(* CoDeSys 2.3.9.59 project: ProgettoSFC.pro *)
(* Libraries: STANDARD.LIB, Iecsfc.lib 12.5.98 11:03:00 *)

(* Task configuration *)
TASK Standard (PRIORITY := 0, INTERVAL := T#10ms);
	MAIN
END_TASK

(* Data type *)
TYPE ALTEZZA: (nd_A, basso, alto);
END_TYPE

(* Data type *)
TYPE COLORE: (nd_C, rosso, altro);
END_TYPE

(* Data type *)
TYPE LOCK_INGRESSO_GIOSTRA :
STRUCT
  FlagNastro: BOOL:=FALSE;
  FlagGIostra: BOOL:=FALSE;
  Turno: TURNO;
END_STRUCT
END_TYPE

(* Data type *)
TYPE PEZZO :
STRUCT
	Colore :COLORE;
	Altezza :ALTEZZA;
END_STRUCT
END_TYPE

(* Data type *)
TYPE POSTO :
STRUCT
	Presenza :BOOL;
	Pezzo :PEZZO;
	Ready :BOOL; (*uguale a 1 quando nel posto è terminato il lavoro*)
	Fine_Lavorazione :BOOL;
END_STRUCT
END_TYPE

(* Data type *)
TYPE TURNO : (Giostr, nastro);
END_TYPE

(* POU MAIN, SFC *)
PROGRAM MAIN
VAR

(*Variabili Pistone*)
  Presenza_Pezzo AT %IX0.0: BOOL;
  Pistone_Indietro AT %IX0.4: BOOL;
  Pistone_Avanti AT %IX0.2: BOOL;
  Pistone_On AT %QX0.2: BOOL;

(*Variabili nastro*)
  Nastro_On AT %QX0.0: BOOL;
  Fine_Corsa AT %IX0.6: BOOL;
  NumPeN: INT:= 0;

(*Variabili gestione timers per non creare conflitti tra nastro pistone e giostra*)
  TimerNP: TON;
  Timer_GN: TON;
  Timer_Nastro: TON;
  ResetTimer: BOOL := FALSE;
  AttesaNP: TIME:= t#0.6s;
  Q: BOOL;
  Delay_Pistone: TON;
  Ritardo_Pistone: BOOL;


(*Interfaccia Nastro-Giostra*)
  InserimentoNG: BOOL:=FALSE; (*Il nastro deve mettere a TRUE quando sta inserendo un pezzo all'interno della giostra e a FALSE quando non lo sta facendo*)
  FineInserimentoGN: BOOL;
  NReady: BOOL := TRUE;    (*Vero quando il nastro autorizza il pistone a spingere un nuovo pezzo*)
  GStart: BOOL := TRUE;    (*Vero quando la giostra è autorizzata a girare*)


(*variabili giostra*)
  Movimento_Giostra AT %QX3.4: BOOL;
  Giostra_BUSY AT %IX6.1: BOOL;
  Giostra: ARRAY[0..7] OF POSTO; (*Array che descrive lo stato di tutti i posti della giostra*)
  TEMP: ARRAY[0..7] OF BOOL; (*Array di supporto per verificare delle condizioni su array di 8 elementi*)
  presenza_fine_lav: BOOL; (*Variabile che deve essere settata a TRUE quando tutti i pezzi presenti nella giostra hanno finito la lavorazione oppure non è presente nessun pezzo nella giostra*)
  i: INT:=0; (*Contatore per il numero di movimenti della giostra (8 movimenti = un giro)*)
  index: INT; (*Variabile di supporto per iterare sull'array*)

  Sensore_Colore AT %IX2.1: BOOL;

  Trapano_Basso AT %IX2.5: BOOL := FALSE;
  TrapanoOn AT %QX3.7:BOOL;
  TimerTrapano: TON; (*timer che tiene conto del tempo di lavorazione trascorso per il pezzo sotto al trapano*)
  FineTrapanazione: BOOL := FALSE;
  Trapano_Alto AT %IX2.3: BOOL;
  Trapano_Down AT %QX7.0: BOOL;

  Tastatore_Basso AT %IX5.3: BOOL;
  Tastatore_Alto AT %IX2.7: BOOL;
  Tastatore_Down AT %QX3.6: BOOL := FALSE;
  ValTastatore: REAL; (*Valore di output del tastatore*)

  Pennarello_Down AT %QX3.3: BOOL;
  Pennarello_Alto AT %IX5.4: BOOL;
  Pennarello_Basso AT %IX5.5: BOOL;
  Fine_Colorazione: BOOL;

  Pistone_PT5_On AT %QX3.1:BOOL := FALSE;
  Pistone_PT5_Avanti AT %IX5.0: BOOL;
  Pistone_PT5_Indietro AT %IX5.1: BOOL;

  Pistone_PT6_On AT%QX3.5: BOOL := FALSE;
  Pistone_PT6_Avanti AT %IX5.7: BOOL;
  Pistone_PT6_Indietro AT %IX5.6: BOOL;
  Pezzo_Baia AT %IX5.2: BOOL;

END_VAR
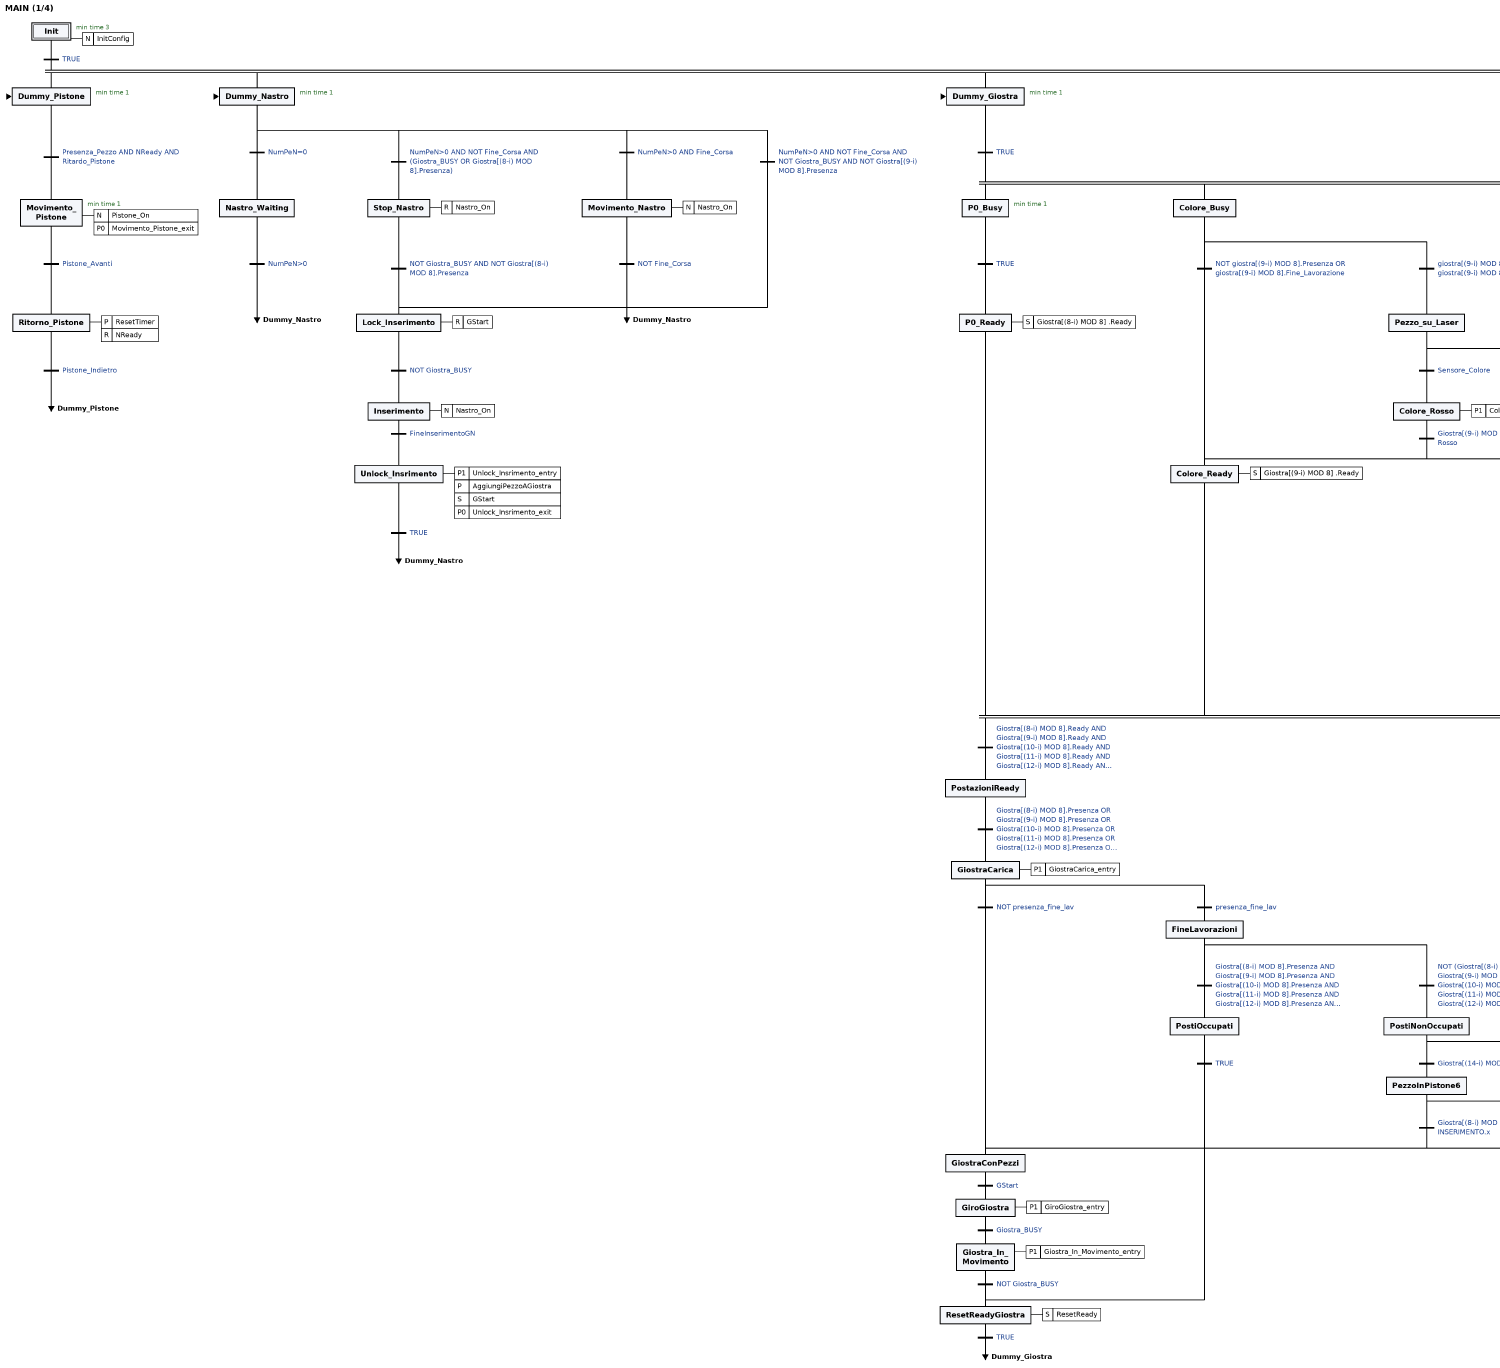
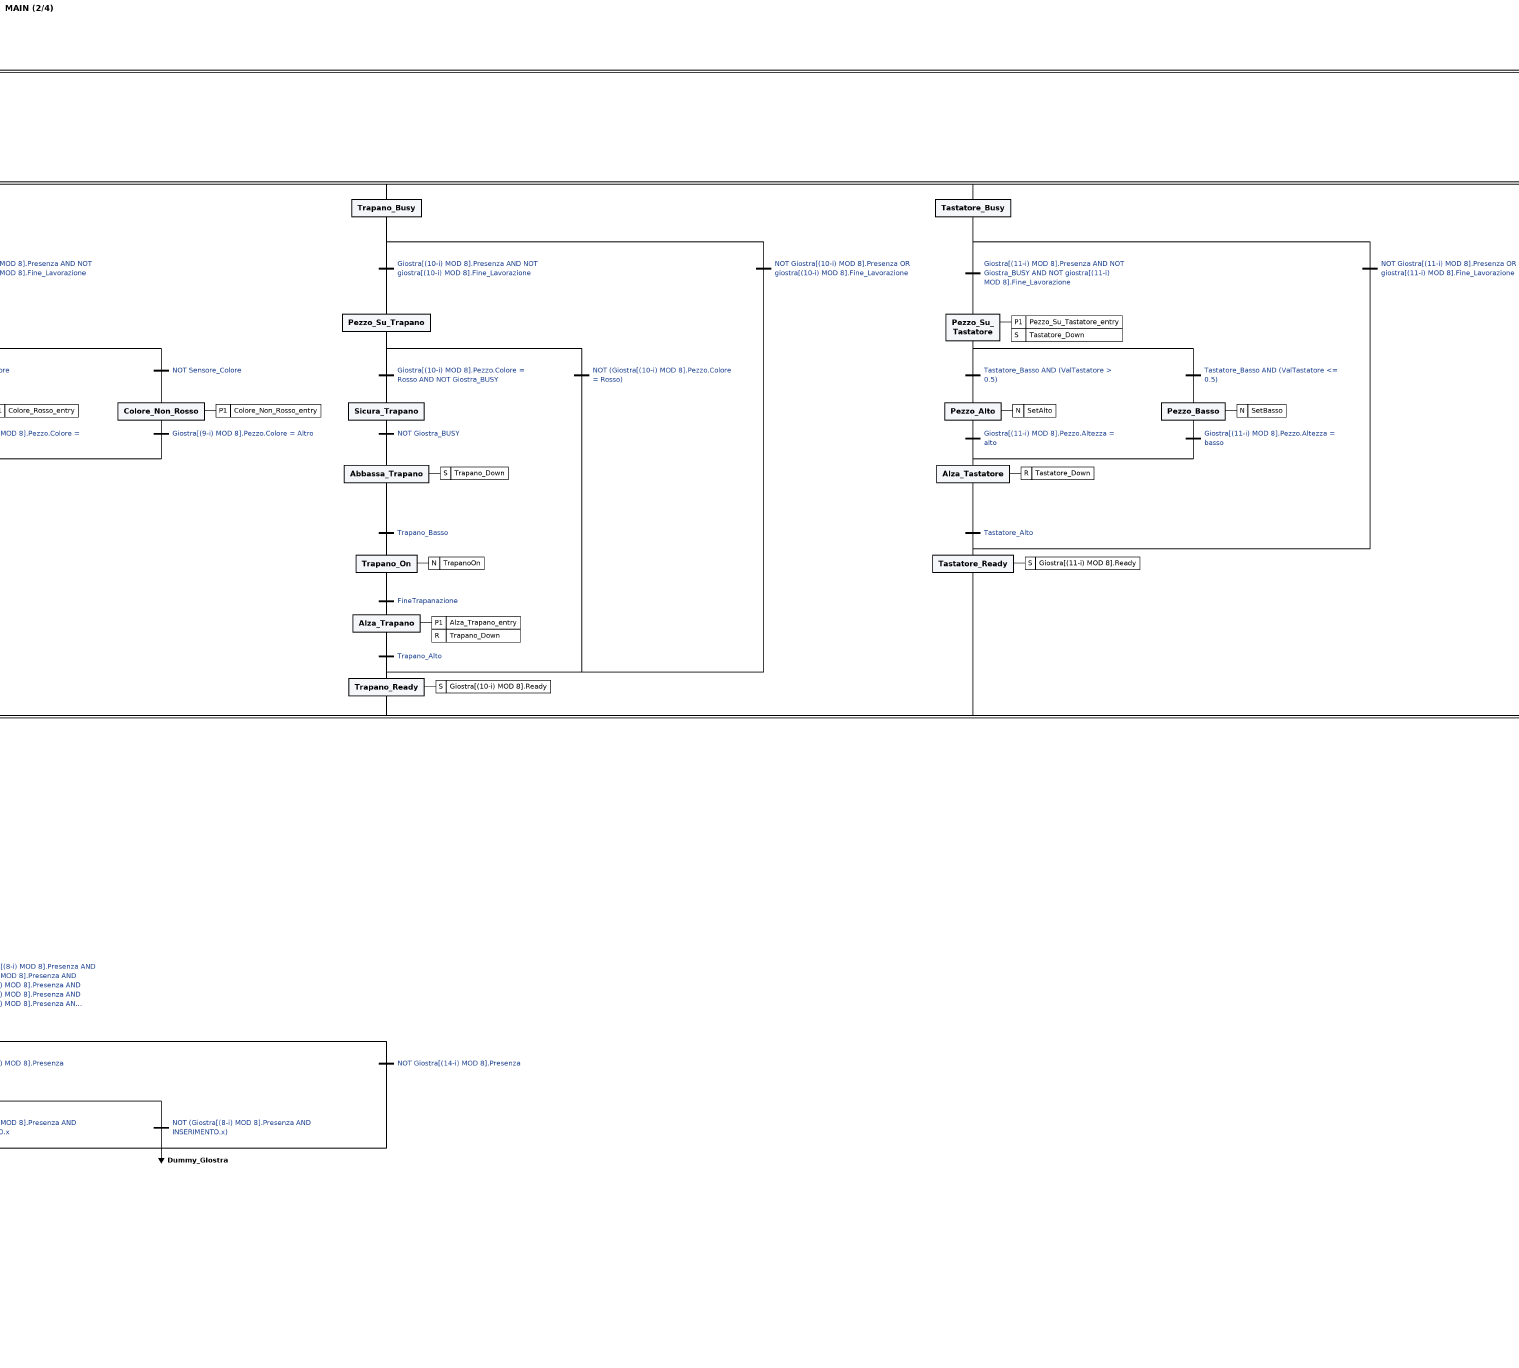
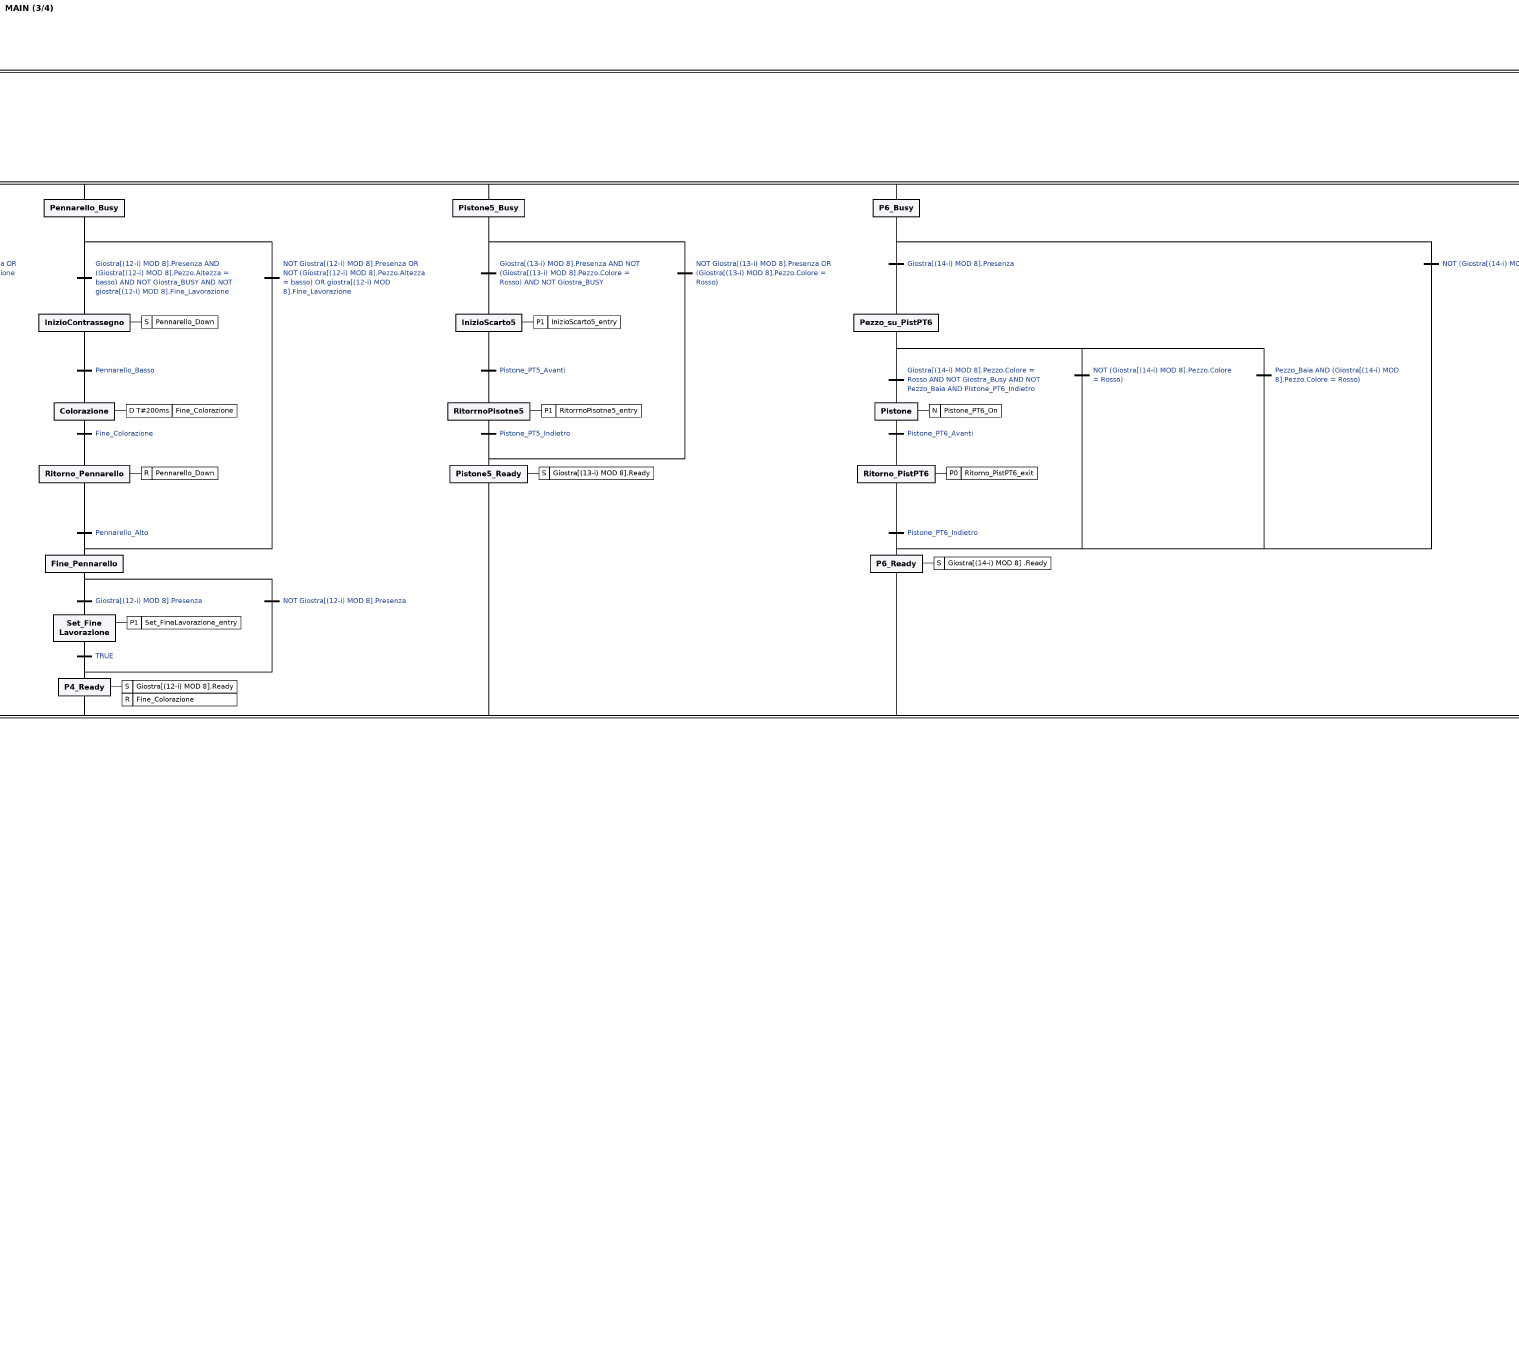
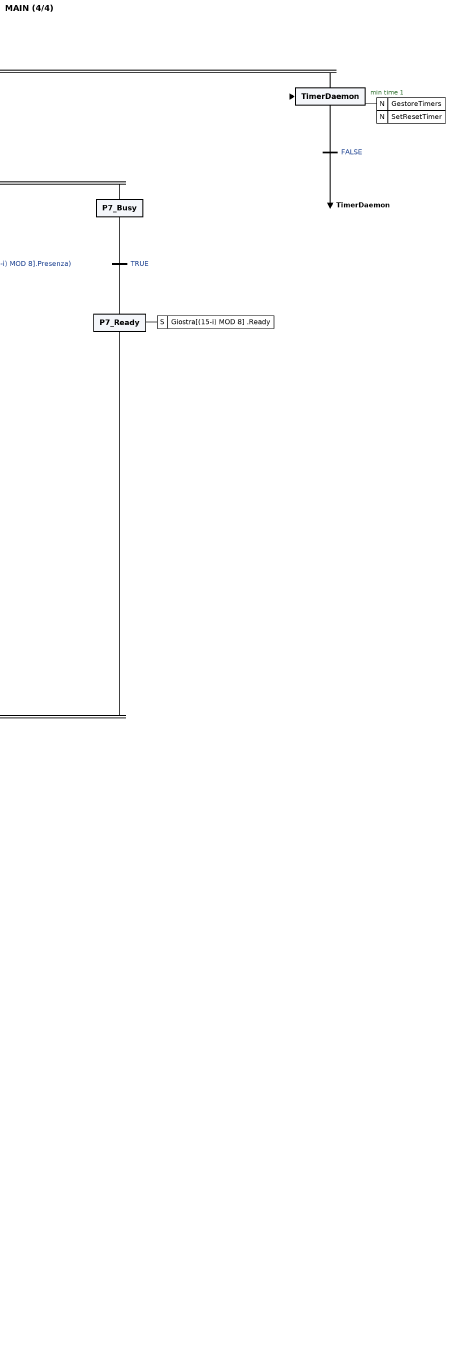
INITIAL_STEP Init: (* min time 3 *)
	InitConfig(N);
END_STEP
TRANSITION FROM Init TO (Dummy_Pistone, Dummy_Nastro, Dummy_Giostra, TimerDaemon) := TRUE;
END_TRANSITION
STEP Dummy_Pistone: (* min time 1 *)
END_STEP
TRANSITION FROM Dummy_Pistone TO Movimento_Pistone := Presenza_Pezzo AND NReady AND Ritardo_Pistone;
END_TRANSITION
STEP Movimento_Pistone: (* min time 1 *)
	Pistone_On(N);
	Movimento_Pistone_exit(P0);
END_STEP
TRANSITION FROM Movimento_Pistone TO Ritorno_Pistone := Pistone_Avanti;
END_TRANSITION
STEP Ritorno_Pistone:
	ResetTimer(P);
	NReady(R);
END_STEP
TRANSITION FROM Ritorno_Pistone TO Dummy_Pistone := Pistone_Indietro;
END_TRANSITION
STEP Dummy_Nastro: (* min time 1 *)
END_STEP
TRANSITION FROM Dummy_Nastro TO Nastro_Waiting := NumPeN=0;
END_TRANSITION
TRANSITION FROM Dummy_Nastro TO Stop_Nastro := NumPeN>0 AND NOT Fine_Corsa AND (Giostra_BUSY OR Giostra[(8-i) MOD 8].Presenza);
END_TRANSITION
TRANSITION FROM Dummy_Nastro TO Movimento_Nastro := NumPeN>0 AND Fine_Corsa;
END_TRANSITION
TRANSITION FROM Dummy_Nastro TO Lock_Inserimento := NumPeN>0 AND NOT Fine_Corsa AND NOT Giostra_BUSY AND NOT Giostra[(9-i) MOD 8].Presenza;
END_TRANSITION
STEP Nastro_Waiting:
END_STEP
TRANSITION FROM Nastro_Waiting TO Dummy_Nastro := NumPeN>0;
END_TRANSITION
STEP Stop_Nastro:
	Nastro_On(R);
END_STEP
TRANSITION FROM Stop_Nastro TO Lock_Inserimento := NOT Giostra_BUSY AND NOT Giostra[(8-i) MOD 8].Presenza;
END_TRANSITION
STEP Movimento_Nastro:
	Nastro_On(N);
END_STEP
TRANSITION FROM Movimento_Nastro TO Dummy_Nastro := NOT Fine_Corsa;
END_TRANSITION
STEP Lock_Inserimento:
	GStart(R);
END_STEP
TRANSITION FROM Lock_Inserimento TO Inserimento := NOT Giostra_BUSY;
END_TRANSITION
STEP Inserimento:
	Nastro_On(N);
END_STEP
TRANSITION FROM Inserimento TO Unlock_Insrimento := FineInserimentoGN;
END_TRANSITION
STEP Unlock_Insrimento:
	Unlock_Insrimento_entry(P1);
	AggiungiPezzoAGiostra(P);
	GStart(S);
	Unlock_Insrimento_exit(P0);
END_STEP
TRANSITION FROM Unlock_Insrimento TO Dummy_Nastro := TRUE;
END_TRANSITION
STEP Dummy_Giostra: (* min time 1 *)
END_STEP
TRANSITION FROM Dummy_Giostra TO (P0_Busy, Colore_Busy, Trapano_Busy, Tastatore_Busy, Pennarello_Busy, Pistone5_Busy, P6_Busy, P7_Busy) := TRUE;
END_TRANSITION
STEP P0_Busy: (* min time 1 *)
END_STEP
TRANSITION FROM P0_Busy TO P0_Ready := TRUE;
END_TRANSITION
STEP P0_Ready:
	Giostra[(8-i) MOD 8] .Ready(S);
END_STEP
STEP Colore_Busy:
END_STEP
TRANSITION FROM Colore_Busy TO Colore_Ready := NOT giostra[(9-i) MOD 8].Presenza OR giostra[(9-i) MOD 8].Fine_Lavorazione;
END_TRANSITION
TRANSITION FROM Colore_Busy TO Pezzo_su_Laser := giostra[(9-i) MOD 8].Presenza AND NOT giostra[(9-i) MOD 8].Fine_Lavorazione;
END_TRANSITION
STEP Pezzo_su_Laser:
END_STEP
TRANSITION FROM Pezzo_su_Laser TO Colore_Rosso := Sensore_Colore;
END_TRANSITION
TRANSITION FROM Pezzo_su_Laser TO Colore_Non_Rosso := NOT Sensore_Colore;
END_TRANSITION
STEP Colore_Rosso:
	Colore_Rosso_entry(P1);
END_STEP
TRANSITION FROM Colore_Rosso TO Colore_Ready := Giostra[(9-i) MOD 8].Pezzo.Colore = Rosso;
END_TRANSITION
STEP Colore_Non_Rosso:
	Colore_Non_Rosso_entry(P1);
END_STEP
TRANSITION FROM Colore_Non_Rosso TO Colore_Ready := Giostra[(9-i) MOD 8].Pezzo.Colore = Altro;
END_TRANSITION
STEP Colore_Ready:
	Giostra[(9-i) MOD 8] .Ready(S);
END_STEP
STEP Trapano_Busy:
END_STEP
TRANSITION FROM Trapano_Busy TO Pezzo_Su_Trapano := Giostra[(10-i) MOD 8].Presenza AND NOT giostra[(10-i) MOD 8].Fine_Lavorazione;
END_TRANSITION
TRANSITION FROM Trapano_Busy TO Trapano_Ready := NOT Giostra[(10-i) MOD 8].Presenza OR giostra[(10-i) MOD 8].Fine_Lavorazione;
END_TRANSITION
STEP Pezzo_Su_Trapano:
END_STEP
TRANSITION FROM Pezzo_Su_Trapano TO Sicura_Trapano := Giostra[(10-i) MOD 8].Pezzo.Colore = Rosso AND NOT Giostra_BUSY;
END_TRANSITION
TRANSITION FROM Pezzo_Su_Trapano TO Trapano_Ready := NOT (Giostra[(10-i) MOD 8].Pezzo.Colore = Rosso);
END_TRANSITION
STEP Sicura_Trapano:
END_STEP
TRANSITION FROM Sicura_Trapano TO Abbassa_Trapano := NOT Giostra_BUSY;
END_TRANSITION
STEP Abbassa_Trapano:
	Trapano_Down(S);
END_STEP
TRANSITION FROM Abbassa_Trapano TO Trapano_On := Trapano_Basso;
END_TRANSITION
STEP Trapano_On:
	TrapanoOn(N);
END_STEP
TRANSITION FROM Trapano_On TO Alza_Trapano := FineTrapanazione;
END_TRANSITION
STEP Alza_Trapano:
	Alza_Trapano_entry(P1);
	Trapano_Down(R);
END_STEP
TRANSITION FROM Alza_Trapano TO Trapano_Ready := Trapano_Alto;
END_TRANSITION
STEP Trapano_Ready:
	Giostra[(10-i) MOD 8].Ready(S);
END_STEP
STEP Tastatore_Busy:
END_STEP
TRANSITION FROM Tastatore_Busy TO Pezzo_Su_Tastatore := Giostra[(11-i) MOD 8].Presenza AND NOT Giostra_BUSY AND NOT giostra[(11-i) MOD 8].Fine_Lavorazione;
END_TRANSITION
TRANSITION FROM Tastatore_Busy TO Tastatore_Ready := NOT Giostra[(11-i) MOD 8].Presenza OR giostra[(11-i) MOD 8].Fine_Lavorazione;
END_TRANSITION
STEP Pezzo_Su_Tastatore:
	Pezzo_Su_Tastatore_entry(P1);
	Tastatore_Down(S);
END_STEP
TRANSITION FROM Pezzo_Su_Tastatore TO Pezzo_Alto := Tastatore_Basso AND (ValTastatore > 0.5);
END_TRANSITION
TRANSITION FROM Pezzo_Su_Tastatore TO Pezzo_Basso := Tastatore_Basso AND (ValTastatore <= 0.5);
END_TRANSITION
STEP Pezzo_Alto:
	SetAlto(N);
END_STEP
TRANSITION FROM Pezzo_Alto TO Alza_Tastatore := Giostra[(11-i) MOD 8].Pezzo.Altezza = alto;
END_TRANSITION
STEP Pezzo_Basso:
	SetBasso(N);
END_STEP
TRANSITION FROM Pezzo_Basso TO Alza_Tastatore := Giostra[(11-i) MOD 8].Pezzo.Altezza = basso;
END_TRANSITION
STEP Alza_Tastatore:
	Tastatore_Down(R);
END_STEP
TRANSITION FROM Alza_Tastatore TO Tastatore_Ready := Tastatore_Alto;
END_TRANSITION
STEP Tastatore_Ready:
	Giostra[(11-i) MOD 8].Ready(S);
END_STEP
STEP Pennarello_Busy:
END_STEP
TRANSITION FROM Pennarello_Busy TO InizioContrassegno := Giostra[(12-i) MOD 8].Presenza AND (Giostra[(12-i) MOD 8].Pezzo.Altezza = basso) AND NOT Giostra_BUSY AND NOT giostra[(12-i) MOD 8].Fine_Lavorazione;
END_TRANSITION
TRANSITION FROM Pennarello_Busy TO Fine_Pennarello := NOT Giostra[(12-i) MOD 8].Presenza OR NOT (Giostra[(12-i) MOD 8].Pezzo.Altezza = basso) OR giostra[(12-i) MOD 8].Fine_Lavorazione;
END_TRANSITION
STEP InizioContrassegno:
	Pennarello_Down(S);
END_STEP
TRANSITION FROM InizioContrassegno TO Colorazione := Pennarello_Basso;
END_TRANSITION
STEP Colorazione:
	Fine_Colorazione(D, T#200ms);
END_STEP
TRANSITION FROM Colorazione TO Ritorno_Pennarello := Fine_Colorazione;
END_TRANSITION
STEP Ritorno_Pennarello:
	Pennarello_Down(R);
END_STEP
TRANSITION FROM Ritorno_Pennarello TO Fine_Pennarello := Pennarello_Alto;
END_TRANSITION
STEP Fine_Pennarello:
END_STEP
TRANSITION FROM Fine_Pennarello TO Set_FineLavorazione := Giostra[(12-i) MOD 8].Presenza;
END_TRANSITION
TRANSITION FROM Fine_Pennarello TO P4_Ready := NOT Giostra[(12-i) MOD 8].Presenza;
END_TRANSITION
STEP Set_FineLavorazione:
	Set_FineLavorazione_entry(P1);
END_STEP
TRANSITION FROM Set_FineLavorazione TO P4_Ready := TRUE;
END_TRANSITION
STEP P4_Ready:
	Giostra[(12-i) MOD 8].Ready(S);
	Fine_Colorazione(R);
END_STEP
STEP Pistone5_Busy:
END_STEP
TRANSITION FROM Pistone5_Busy TO InizioScarto5 := Giostra[(13-i) MOD 8].Presenza AND NOT (Giostra[(13-i) MOD 8].Pezzo.Colore = Rosso) AND NOT Giostra_BUSY;
END_TRANSITION
TRANSITION FROM Pistone5_Busy TO Pistone5_Ready := NOT Giostra[(13-i) MOD 8].Presenza OR (Giostra[(13-i) MOD 8].Pezzo.Colore = Rosso);
END_TRANSITION
STEP InizioScarto5:
	InizioScarto5_entry(P1);
END_STEP
TRANSITION FROM InizioScarto5 TO RitorrnoPisotne5 := Pistone_PT5_Avanti;
END_TRANSITION
STEP RitorrnoPisotne5:
	RitorrnoPisotne5_entry(P1);
END_STEP
TRANSITION FROM RitorrnoPisotne5 TO Pistone5_Ready := Pistone_PT5_Indietro;
END_TRANSITION
STEP Pistone5_Ready:
	Giostra[(13-i) MOD 8].Ready(S);
END_STEP
STEP P6_Busy:
END_STEP
TRANSITION FROM P6_Busy TO Pezzo_su_PistPT6 := Giostra[(14-i) MOD 8].Presenza;
END_TRANSITION
TRANSITION FROM P6_Busy TO P6_Ready := NOT (Giostra[(14-i) MOD 8].Presenza);
END_TRANSITION
STEP Pezzo_su_PistPT6:
END_STEP
TRANSITION FROM Pezzo_su_PistPT6 TO Pistone := Giostra[(14-i) MOD 8].Pezzo.Colore = Rosso AND NOT Giostra_Busy AND NOT Pezzo_Baia AND Pistone_PT6_Indietro;
END_TRANSITION
TRANSITION FROM Pezzo_su_PistPT6 TO P6_Ready := NOT (Giostra[(14-i) MOD 8].Pezzo.Colore = Rosso);
END_TRANSITION
TRANSITION FROM Pezzo_su_PistPT6 TO P6_Ready := Pezzo_Baia AND (Giostra[(14-i) MOD 8].Pezzo.Colore = Rosso);
END_TRANSITION
STEP Pistone:
	Pistone_PT6_On(N);
END_STEP
TRANSITION FROM Pistone TO Ritorno_PistPT6 := Pistone_PT6_Avanti;
END_TRANSITION
STEP Ritorno_PistPT6:
	Ritorno_PistPT6_exit(P0);
END_STEP
TRANSITION FROM Ritorno_PistPT6 TO P6_Ready := Pistone_PT6_Indietro;
END_TRANSITION
STEP P6_Ready:
	Giostra[(14-i) MOD 8] .Ready(S);
END_STEP
STEP P7_Busy:
END_STEP
TRANSITION FROM P7_Busy TO P7_Ready := TRUE;
END_TRANSITION
STEP P7_Ready:
	Giostra[(15-i) MOD 8] .Ready(S);
END_STEP
TRANSITION FROM (P0_Ready, Colore_Ready, Trapano_Ready, Tastatore_Ready, P4_Ready, Pistone5_Ready, P6_Ready, P7_Ready) TO PostazioniReady := Giostra[(8-i) MOD 8].Ready AND Giostra[(9-i) MOD 8].Ready AND Giostra[(10-i) MOD 8].Ready AND Giostra[(11-i) MOD 8].Ready AND Giostra[(12-i) MOD 8].Ready AND Giostra[(13-i) MOD 8].Ready AND Giostra[(14-i) MOD 8].Ready AND Giostra[(15-i) MOD 8].Ready;
END_TRANSITION
STEP PostazioniReady:
END_STEP
TRANSITION FROM PostazioniReady TO GiostraCarica := Giostra[(8-i) MOD 8].Presenza OR Giostra[(9-i) MOD 8].Presenza OR Giostra[(10-i) MOD 8].Presenza OR Giostra[(11-i) MOD 8].Presenza OR Giostra[(12-i) MOD 8].Presenza OR Giostra[(13-i) MOD 8].Presenza OR Giostra[(14-i) MOD 8].Presenza OR Giostra[(15-i) MOD 8].Presenza;
END_TRANSITION
STEP GiostraCarica:
	GiostraCarica_entry(P1);
END_STEP
TRANSITION FROM GiostraCarica TO GiostraConPezzi := NOT presenza_fine_lav;
END_TRANSITION
TRANSITION FROM GiostraCarica TO FineLavorazioni := presenza_fine_lav;
END_TRANSITION
STEP FineLavorazioni:
END_STEP
TRANSITION FROM FineLavorazioni TO PostiOccupati := Giostra[(8-i) MOD 8].Presenza AND Giostra[(9-i) MOD 8].Presenza AND Giostra[(10-i) MOD 8].Presenza AND Giostra[(11-i) MOD 8].Presenza AND Giostra[(12-i) MOD 8].Presenza AND Giostra[(13-i) MOD 8].Presenza AND Giostra[(14-i) MOD 8].Presenza AND Giostra[(15-i) MOD 8].Presenza;
END_TRANSITION
TRANSITION FROM FineLavorazioni TO PostiNonOccupati := NOT (Giostra[(8-i) MOD 8].Presenza AND Giostra[(9-i) MOD 8].Presenza AND Giostra[(10-i) MOD 8].Presenza AND Giostra[(11-i) MOD 8].Presenza AND Giostra[(12-i) MOD 8].Presenza AND Giostra[(13-i) MOD 8].Presenza AND Giostra[(14-i) MOD 8].Presenza AND Giostra[(15-i) MOD 8].Presenza);
END_TRANSITION
STEP PostiOccupati:
END_STEP
TRANSITION FROM PostiOccupati TO ResetReadyGiostra := TRUE;
END_TRANSITION
STEP PostiNonOccupati:
END_STEP
TRANSITION FROM PostiNonOccupati TO PezzoInPistone6 := Giostra[(14-i) MOD 8].Presenza;
END_TRANSITION
TRANSITION FROM PostiNonOccupati TO GiostraConPezzi := NOT Giostra[(14-i) MOD 8].Presenza;
END_TRANSITION
STEP PezzoInPistone6:
END_STEP
TRANSITION FROM PezzoInPistone6 TO GiostraConPezzi := Giostra[(8-i) MOD 8].Presenza AND INSERIMENTO.x;
END_TRANSITION
TRANSITION FROM PezzoInPistone6 TO Dummy_GIostra := NOT (Giostra[(8-i) MOD 8].Presenza AND INSERIMENTO.x);
END_TRANSITION
STEP GiostraConPezzi:
END_STEP
TRANSITION FROM GiostraConPezzi TO GiroGiostra := GStart;
END_TRANSITION
STEP GiroGiostra:
	GiroGiostra_entry(P1);
END_STEP
TRANSITION FROM GiroGiostra TO Giostra_In_Movimento := Giostra_BUSY;
END_TRANSITION
STEP Giostra_In_Movimento:
	Giostra_In_Movimento_entry(P1);
END_STEP
TRANSITION FROM Giostra_In_Movimento TO ResetReadyGiostra := NOT Giostra_BUSY;
END_TRANSITION
STEP ResetReadyGiostra:
	ResetReady(S);
END_STEP
TRANSITION FROM ResetReadyGiostra TO Dummy_Giostra := TRUE;
END_TRANSITION
STEP TimerDaemon: (* min time 1 *)
	GestoreTimers(N);
	SetResetTimer(N);
END_STEP
TRANSITION FROM TimerDaemon TO TimerDaemon := FALSE;
END_TRANSITION

ACTION Movimento_Pistone_exit:
NumPeN := NumPeN + 1;
END_ACTION

ACTION Unlock_Insrimento_entry:
FineInserimentoGN := FALSE;
END_ACTION

ACTION Unlock_Insrimento_exit:
NumPeN := NumPeN - 1;
END_ACTION

ACTION Colore_Rosso_entry:
giostra[(9-i) MOD 8].Pezzo.Colore := rosso;
END_ACTION

ACTION Colore_Non_Rosso_entry:
giostra[(9-i) MOD 8].Pezzo.Colore := altro;
END_ACTION

ACTION Alza_Trapano_entry:
FineTrapanazione := FALSE;
END_ACTION

ACTION Pezzo_Su_Tastatore_entry:
IF (i MOD 2) = 1 THEN
    ValTastatore := 0.6;
	ELSE
    		ValTastatore := 0.4;
END_IF;
END_ACTION

ACTION Set_FineLavorazione_entry:
Giostra[(12-i) MOD 8].Fine_Lavorazione := TRUE;
END_ACTION

ACTION InizioScarto5_entry:
Pistone_PT5_On := TRUE;
END_ACTION

ACTION RitorrnoPisotne5_entry:
Giostra[(13-i) MOD 8].Presenza:= FALSE;
Giostra[(13-i) MOD 8].Pezzo.Altezza := nd_a;
Giostra[(13-i) MOD 8].Pezzo.Colore := nd_c;
Giostra[(13-i) MOD 8].Fine_Lavorazione:=FALSE;

Pistone_PT5_On := FALSE;
END_ACTION

ACTION Ritorno_PistPT6_exit:
Giostra[(14-i) MOD 8].Presenza := FALSE;
Giostra[(14-i) MOD 8].Fine_Lavorazione := FALSE;
Giostra[(14-i) MOD 8].Pezzo.Altezza := nd_A;
Giostra[(14-i) MOD 8].Pezzo.Colore := nd_C;
END_ACTION

ACTION GiostraCarica_entry:
FOR index := 0 TO 7 BY 1 DO
 	IF (NOT Giostra[index].Presenza OR Giostra[index].Fine_Lavorazione) THEN
	TEMP[index] := TRUE;
    	ELSE
       		TEMP[index] := FALSE;
  	END_IF;
END_FOR;

IF (TEMP[0] AND TEMP[1] AND TEMP[2] AND TEMP[3] AND TEMP[4] AND TEMP[5] AND TEMP[6] AND TEMP[7]) THEN
  	presenza_fine_lav := TRUE;
  	ELSE
    		presenza_fine_lav :=FALSE;
END_IF
END_ACTION

ACTION GiroGiostra_entry:
Movimento_Giostra := TRUE;
END_ACTION

ACTION Giostra_In_Movimento_entry:
IF i=7 THEN
    i:=0;
	ELSE
  	 i := i + 1;
END_IF;

Movimento_Giostra := FALSE;
END_ACTION
END_PROGRAM
ACTION AggiungiPezzoAGiostra:
Giostra[(8-i) MOD 8].Presenza := TRUE;
Giostra[(8-i) MOD 8].Ready :=TRUE;
END_ACTION
ACTION GestoreTimers:
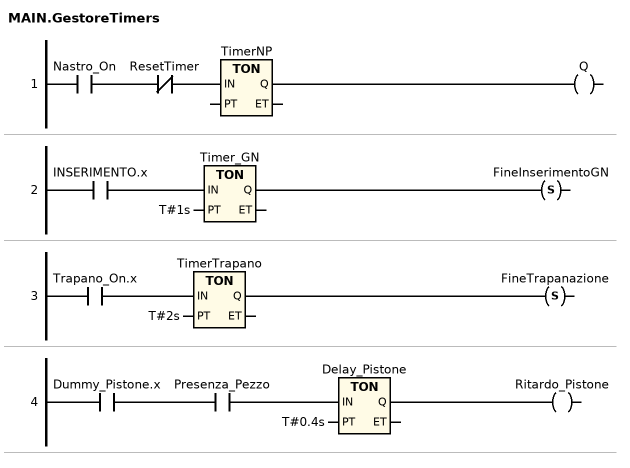
_LD_ (* Ladder Diagram *)
NETWORK 1
	[Nastro_On] - [/ResetTimer] - TimerNP:TON(IN: *, PT: ) --- (Q)
NETWORK 2
	[INSERIMENTO.x] - Timer_GN:TON(IN: *, PT:  T#1s) --- (S FineInserimentoGN)
NETWORK 3
	[Trapano_On.x] - TimerTrapano:TON(IN: *, PT: T#2s) --- (S FineTrapanazione)
NETWORK 4
	[Dummy_Pistone.x] - [Presenza_Pezzo] - Delay_Pistone:TON(IN: *, PT: T#0.4s) --- (Ritardo_Pistone)
_END_LD_
(* the same logic as Structured Text *)
(* Network 1: see the listing above *)
(* Network 2 *)
Timer_GN(IN := INSERIMENTO.x, PT :=  T#1s);
IF Timer_GN.Q THEN FineInserimentoGN := TRUE; END_IF;
(* Network 3 *)
TimerTrapano(IN := Trapano_On.x, PT := T#2s);
IF TimerTrapano.Q THEN FineTrapanazione := TRUE; END_IF;
(* Network 4 *)
Delay_Pistone(IN := Dummy_Pistone.x AND Presenza_Pezzo, PT := T#0.4s);
Ritardo_Pistone := Delay_Pistone.Q;
END_ACTION
ACTION InitConfig:
TimerNP.PT := t#20d;
NReady := TRUE;
END_ACTION
ACTION ResetReady:
FOR index := 0 TO 7 BY 1 DO
   Giostra[index].Ready := FALSE;
END_FOR;
END_ACTION
ACTION SetAlto:
Giostra[(11-i) MOD 8].Pezzo.Altezza := alto;
END_ACTION
ACTION SetBasso:
Giostra[(11-i) MOD 8].Pezzo.Altezza := basso;
END_ACTION
ACTION SetResetTimer:
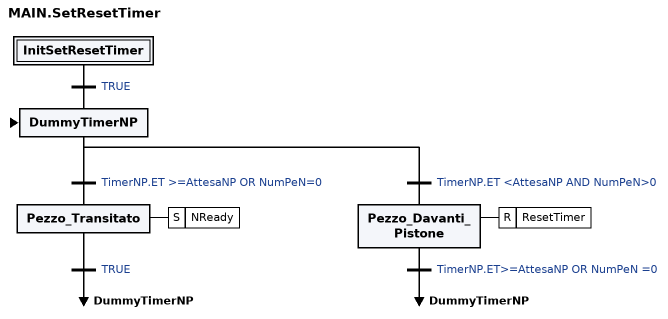
INITIAL_STEP InitSetResetTimer:
END_STEP
TRANSITION FROM InitSetResetTimer TO DummyTimerNP := TRUE;
END_TRANSITION
STEP DummyTimerNP:
END_STEP
TRANSITION FROM DummyTimerNP TO Pezzo_Transitato := TimerNP.ET >=AttesaNP OR NumPeN=0;
END_TRANSITION
TRANSITION FROM DummyTimerNP TO Pezzo_Davanti_Pistone := TimerNP.ET <AttesaNP AND NumPeN>0;
END_TRANSITION
STEP Pezzo_Davanti_Pistone:
	ResetTimer(R);
END_STEP
TRANSITION FROM Pezzo_Davanti_Pistone TO DummyTimerNP := TimerNP.ET>=AttesaNP OR NumPeN =0;
END_TRANSITION
STEP Pezzo_Transitato:
	NReady(S);
END_STEP
TRANSITION FROM Pezzo_Transitato TO DummyTimerNP := TRUE;
END_TRANSITION
END_ACTION
